TYPE DUT_ALM :
STRUCT
	GeneralFailure: BOOL;
	TimeFailure: BOOL;
	InAlarm: BOOL := TimeFailure OR GeneralFailure;
END_STRUCT
END_TYPE

(* stored: Version 1.1.0.1, ProductVersion 3.1.4024.12
   DUT DUT_ALM: Id {5d8818e7-c143-44b5-a75f-8d988f63bb22} *)
